Universal Robots PolyScope program: cottonHome.urp

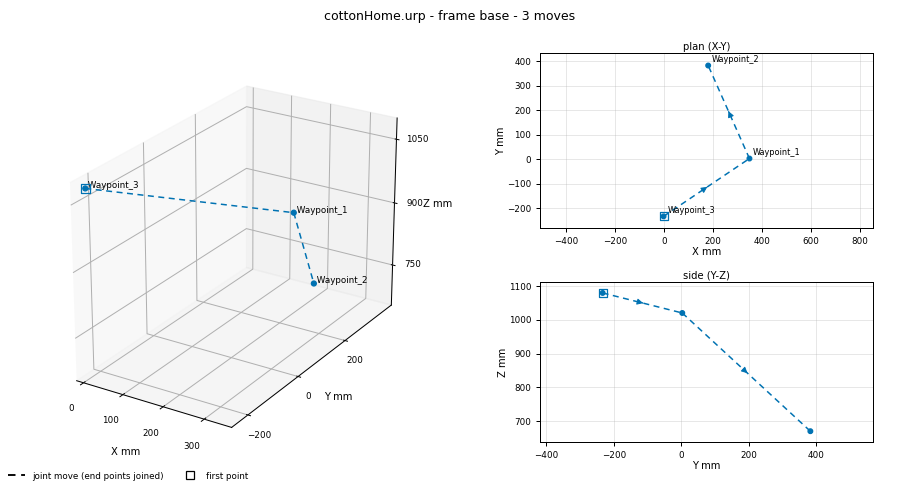
[picture p0: tool path of cottonHome.urp in frame base, 3 of 4 moves have a stored position in this frame; points joined in program order, loops and branches not executed]
Program cottonHome (installation=default directory=/programs/DavidMelin createdIn=5.12.4.1101661 lastSavedIn=5.12.4.1101661 robotSerialNumber=20225502378)
Calibrated DH parameters: a=[0.00022, -0.425328, -0.389701, 0.000059, 0.000065, 0]; d=[0.162608, 0.803456, 9.992211, -10.662202, 0.099702, 0.099559]; alpha=[1.570756, 0.001543, 0.004316, 1.570651, -1.570122, 0]; deltaTheta=[0, 0.002917, 0.116094, -0.119008, 0, -0.000001]
Robot Program (runOnlyOnce=true)
  URCap Gripper Activate (Robotiq_Grippers, Robotiq Inc.) dataModel(ResetAndActivateKey=false)
  MoveJ speed 60 deg/s, acceleration 80 deg/s^2 (useActiveTCP=true) feature=Base
    Waypoint Waypoint_3: TCP in base x=-1.305 y=-233.152 z=1080.057 mm, rx=-0.0066 ry=-2.2185 rz=2.2186 rad; joints [-0.004, -90, 0.002, -89.998, -0.002, 0] deg
    Waypoint Waypoint_1: TCP in base x=349.126 y=2.769 z=1020.655 mm, rx=-1.2149 ry=1.7206 rz=-2.0946 rad; joints [42.422, -93.623, -24.756, -89.916, 0.048, 0.001] deg
    Waypoint Waypoint_2: TCP in base x=180.817 y=382.289 z=670.407 mm, rx=-2.5356 ry=0.5347 rz=-0.6666 rad; joints [91.157, -74.563, -85.1, -87.865, 57.347, 18.15] deg
    Waypoint Waypoint (Variable): variable=cotonHomePos
